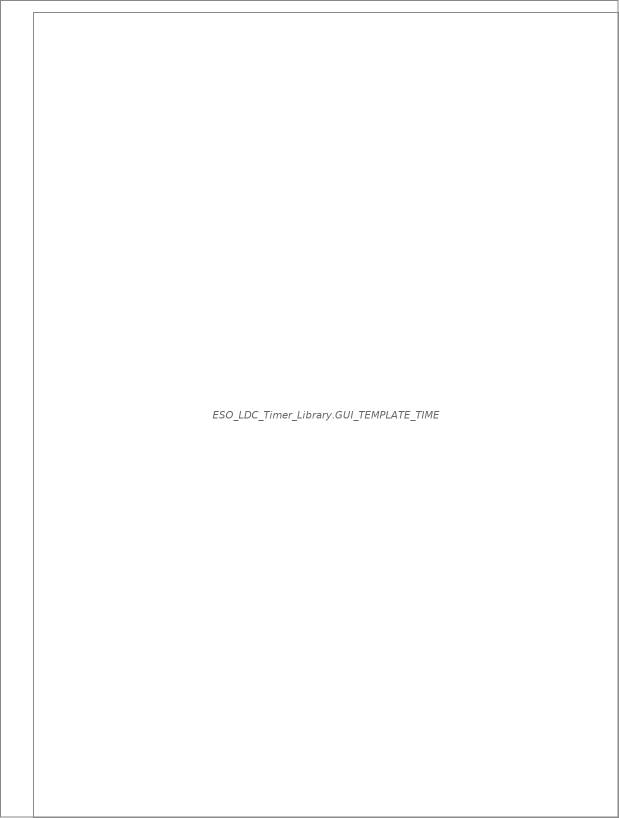
VISUALIZATION GUI_TIMER  // 619x818
    Frame (33,12 586x806)
        shows ESO_LDC_Timer_Library.GUI_TEMPLATE_TIME(m_Instance := MAIN.fbTimer)
END_VISUALIZATION

(* stored: Version 1.1.0.1, ProductVersion 3.1.4024.9
   Visu GUI_TIMER: Id {51fb39e1-872d-4bfb-9c4b-e90ab312902d} *)
